// TIA Portal V17 export
// export: Created 2023-09-10T16:27:53.0486675Z, ExportSetting WithDefaults, DisplayName Totally Integrated Automation Portal, DisplayVersion V17, DisplayName TIA Portal Openness, DisplayVersion V17, DisplayName TIA Portal Version Control Interface, DisplayVersion V17, DisplayName STEP 7 Professional, DisplayVersion V17, DisplayName STEP 7 Safety, DisplayVersion V17, DisplayName WinCC Advanced, DisplayVersion V17
DATA_BLOCK "HMI"   // DB2
{ S7_Optimized_Access := 'FALSE' }
VERSION : 0.1
// stored: AutoNumber true, DBAccessibleFromOPCUA true, IsOnlyStoredInLoadMemory false, IsWriteProtectedInAS false
   VAR RETAIN
      sensor : Bool := 1;
      machinePosition : DInt := 77;
      encoderTurn : DInt := 20;
      encoderPosition : Int;
      setpoint : Int;
      buttonBase : Bool;
      buttonStart : Bool;
      buttonStop : Bool;
      jogBackward : Bool;
      jogForward : Bool;
      jogVelocity : Int := 50;
      machineVelocity : Int := 70;
      baseVelocity : Int := 20;
      machineConst : DInt := 42625;   // numberOfpulseEncoder 1023 numberOfTurnPer90st 2,24*90
      serwisSetpointEnable : Bool;
      serwisMachineSetpoint : DInt;
   END_VAR
BEGIN
END_DATA_BLOCK
